// TIA Portal V16 export
// export: Created 2023-03-29T11:04:36.4873224Z, ExportSetting WithDefaults, DisplayName Totally Integrated Automation Portal, DisplayVersion V16 Update 6, DisplayName TIA Portal Version Control Interface, DisplayVersion V16 Update 2, DisplayName TIA Portal Openness, DisplayVersion V16 Update 6, DisplayName STEP 7 Professional, DisplayVersion V16 Update 6, DisplayName STEP 7 Safety, DisplayVersion V16, DisplayName WinCC Advanced, DisplayVersion V16 Update 6
DATA_BLOCK "db10organizacyjna"   // DB10
TITLE = Instance SCADA
{ S7_Optimized_Access := 'FALSE' }
AUTHOR : RTecmer
VERSION : 0.1
// stored: AutoNumber false, DBAccessibleFromOPCUA true, IsOnlyStoredInLoadMemory false, IsWriteProtectedInAS false
   VAR
      Clock : Time;
      Watchdog : Int;
      insPompa1 : Word;
      insPompa2 : Word;
      insPompa3 : Word;
      insPompa4 : Word;
      instB6_bar_act_miasto : Real;   // Ciśnienie B6 miasto [Real]
      instB5_bar_act_magistrala : Real;   // Ciśnienie B5 magistrala [Real]
      actPozycja_Z10 : Word;   // Aktualna pozycja Z10 [%]
      errorModbusRTU_SCADA : Word;   // awaria modbus rtu falownik bit 0, przepływomierz pompownia bit 1, przepływomierz magistra bit 2, sterownik MT101 bit 3
      HourCounterP1 : DWord;   // Counter Work
      HourCounterP2 : DWord;   // Counter Work
      HourCounterP3 : DWord;   // Counter Work
      HourCounterP4 : DWord;
      TimeHz : Int := 45;
      Time_ONK1 : Int := 110;
      Time_ONK2 : Int := 300;
      Time_OFFK1 : Int := 5;
      Time_OFFK2 : Int := 2;
      "PID_Compact_1_sPid_Cmpt.r_Sp_Hlm" : Real := 2.2;
      "PID_Compact_1_sPid_Cmpt.r_Sp_LIm" : Real := 1.5;
      set_Hz_P1P4 : Real;   // Aktualne Hz na falowniku
      setpoint_SV_bar : Real := 1.8;   // Zadana wartość ciśnienie do PID [bar]
      set_min_press_bar_B8 : Real := 0.0;   // minimalne ciśnienie bezpieczeństwa [bar] B8
      instFlowDN225_act_Q1 : Real;   // aktualny przepływ Q1 pompownia
      reset_modbus_TCP : Bool;   // reset komunikacji modbus TCP
      instB7_bar_act_pompownia : Real := 0.28;   // aktualne
      min_Bar_set : Real := 1.7;   // Minimalne ciśnienie zadane
      max_Bar_set : Real := 2.7;   // Maxymalne ciśnienie zadane
      actTime : Real;   // aktualny czas
      "pos_Setpint_SV bar" : Real;   // Aktualna wartość zadanaego ciśnienie
      act_stanP1 : Int;   // Zmienna na potzrzeby trenów pracy pompy
      act_statnP2 : Int;   // Zmienna na potzrzeby trenów pracy pompy
      act_stanP3 : Int;   // Zmienna na potzrzeby trenów pracy pompy
      act_stanP4 : Int;
      instSumFlowDN225_Q1 : Real;   // Aktualny przepływ na wlocie oczyszczalni m3/h
      switch_ModelSterowania : Word := 1;   // Zmienna przyjmująca wartość dziesiętnią oznaczającą model sterowania
      instB8_bar_act_suchobieg : Real;   // Ciśnienie suchobiegu (0-1bar)
      "alarms only" : Word;   // Instancja alarmów (bit 146.4 - Error Modbus),(bit 146.5-Warning Modbau)
      inverterPomp_Status : Word;   // Status falownika pomp
      inst_act_Current_Inverters : Real;   // Aktualny prąd falownika [A]
      set_press_bar_Max : Real := 7.888;   // Maxymalne dopuszczalne ciśnienie w rurociągu [bar]
      ampere_Max : Real := 56.0;   // Edytowalne - Maxymalne dopuszczalne przeciążenie [A]
      act_Hz_Inverter_1 : Real;   // Aktualne Hz na falowniku
      ins_ModeWorkContactronP1 : Word;   // Zmienna przechowująca informację o stanie napędu (0-postój, 1-falownik, 2-sieć)
      ins_ModeWorkContactronP2 : Word;   // Zmienna przechowująca informację o stanie napędu (0-postój, 1-falownik, 2-sieć)
      ins_ModeWorkContactronP3 : Word;   // Zmienna przechowująca informację o stanie napędu (0-postój, 1-falownik, 2-sieć)
      ins_ModeWorkContactronP4 : Word;   // Zmienna przechowująca informację o stanie napędu (0-postój, 1-falownik, 2-sieć)
      instB9_bar_act_Granica : Real;   // Wartość bar w sterowanym zbiorniku
      PV_HWrn_set_correct : Real := 2.1;   // Wspóczninik służący wprowadzeniu korekty ostrzeżenia przekroczenia wartości zadanej bar
      PV_LWrn_set_correct : Real := 0.6;   // Wspóczninik służący wprowadzeniu korekty ostrzeżenia zbyt niskia wartości bar w stosunku do zadanej
      TimeHistere_set_bar : Int := 1;   // Czas zwłoki przed zmianą bar zadanego podczas redukcji azotu
      avg_bar : Real;   // srednia wartość ciśnienie
      RTU_Fal_1errorStatus : Word;   // Status błędu komunikacji Modbus RTU
      RTU_MPP04_1errorStatus : Word;   // Status błędu komunikacji Modbus RTU
      RTU_MPP04_2errorStatus : Word;   // Status błędu komunikacji Modbus RTU
      RTU_MT101 : Word;   // Status błędu komunikacji Modbus RTU
      RTU_stepRESET : Bool := 1;   // Krok pętli Modbus RTU na potrzeby SCADA (RESET)
      setRTU_Error : Bool;   // Znacznik błedu modbus RTU
      instSecStart_City_1 : Int;   // Sekundy start przetłaczanie
      instSecStop_City_1 : Int;   // Sekundy stop przetłaczanie
      instSecStart_Replen_1 : Int;   // Sekundy start dosilanie
      instSecStop_Replen_1 : Int;   // Sekundy stop dosilanie
      CounterOverTempFa : Int;   // Licznik wystąpienia usterki przegrzania
      instSecStart_Filling_1 : Int;   // Sekundy start napełniania
      instSecStop_Filling_1 : Int;   // Sekundy stop napełniania
      CounterOverVoltFal : Int;   // Licznik wystapienia usterki wysokie VDC
      instHourStart_Filling_1 : Int;   // Godzina start napełniania
      instMinutStart_Filling : Int;   // Minuta start napełniania
      instHourStop_Filling_1 : Int;   // Godzina stop napełniania
      instMinutStopt_Filling : Int;   // Minuta stop napełniania
      instFlowDN500_act_Q2 : Real;   // Aktualna wartośc przepływu Q2 magistrala
      instSumFlowDN500_Q2 : Real;   // Aktualna wartośc sumy przepywu Q2 magistrala
      instHourStart_Filling : DTL;   // Godzina start napełniania
      instHourStop_Filling : DTL;   // Godzina stop napełniania
      instHourStart_City : DTL;   // Godzina start przetłaczanie miasto DN225
      instHourStop_City : DTL;   // Godzina stop przetłaczanie miasto DN225
      instHourStart_Replen : DTL;   // Godzina start dosilanie DN500
      instHourStop_Replen : DTL;   // Godzina stop dosilanie DN500
      actQ1_przepyw_pompownia_Int : Word;   // Aktualny przepływ na Q1 pompownia
      actQ2_przepyw_pompownia_Int : Word;   // Aktualny przepływ na Q2 pompownia
      inst_sum_FlowDN255_act_Q2_int : Word;   // aktualna suma przepływu Q1 (int)
      inst_sumFlowDN500_act_Q2_int : Word;   // aktualna suma przepływu Q2 (int)
      instHourStart_City_1 : Int;   // Godzina start przetłaczanie miasto DN225
      instMinutStart_City : Int;   // Minuty start przetłaczanie miasto DN225
      instHourStop_City_1 : Int;   // Godzina stop przetłaczanie miasto DN225
      instMinutStopt_City : Int;   // Minuty stop przetłaczanie miasto DN225
      instHourStart_Replen_1 : Int;   // Godzina start dosilanie magistrala DN500
      instMinutStart_Replen : Int;   // Minuty start dosilanie magistrala DN500
      instHourStop_Replen_1 : Int;   // Godzina stop dosilanie magistrala DN500
      instMinutStopt_Replen : Int;   // Minuty stop dosilanie magistrala DN500
      instvValveZ1 : Word;   // Zasuwa zbiornik - spust zbiornik 1
      instvValveZ2 : Word;   // Zasuwa zbiornik - zasilanie zbiornik 1
      instvValveZ3 : Word;   // Zasuwa zbiornik - spust zbiornik 2
      instvValveZ4 : Word;   // Zasuwa zbiornik - zasilanie zbiornik 2
      instvValveZ5 : Word;   // Zasuwa zbiornik - spust zbiornik 3
      instvValveZ6 : Word;   // Zasuwa zbiornik - zasilanie zbiornik 3
      instvValveZ7 : Word;   // Zasuwa zbiornik - spust zbiornik 4
      instvValveZ8 : Word;   // Zasuwa zbiornik - zasilanie zbiornik 4
      instvValveZ9 : Word;   // Zasuwa suchobieg
      instvValveZ10 : Word;   // Zasuwa zbiornik regulowana - zasilanie
      actHour : Int;   // Godzina start dosilanie magistrala DN500
      actMinut : Int;   // aktualny czas
      actSec : Int := 0;   // aktualny czas
   END_VAR
BEGIN
END_DATA_BLOCK
